(* CoDeSys 2.3.9.41 project: pns-dio.pro *)
(* Libraries: STANDARD.LIB 4.10.05 10:14:46, IECSFC.LIB 13.4.06 14:51:28, SYSLIBTIME.LIB 20.2.06 13:31:16, SYSTASKINFO.LIB 20.2.06 13:31:38, ANALYZATION.LIB 5.10.99 08:05:06, SYSLIBCALLBACK.LIB 20.2.06 13:31:08 *)

(* PLC configuration (modules and I/O channels)
AT %IB0.0 [ByteInput] 8 discrete inputs
DO0 AT %QX1.0 [BitOutput] relay
DO1 AT %QX2.0 [BitOutput] relay
DO2 AT %QX3.0 [BitOutput] relay
DO3 AT %QX4.0 [BitOutput] relay
DO4 AT %QX5.0 [BitOutput] relay
DO5 AT %QX6.0 [BitOutput] relay
AT %QX7.0 [BitOutput] Special output
RS-485-1 [COM1_USART] node 0, in %IB8.0.0 out %QB8.0.0 {CommunicationSpeed = 19200; Parity = NO PARITY CHECK; BitLength = 8 bits; StopLength = One stop bit; InterfaceType = RS485; FrameOriented = RTU; Timeout = 0; Visibility = No}
DIs AT %QW8.1.0 [WordOutput]
DOs AT %QW8.2.0 [WordOutput]
*)

(* POU PLC_PRG, ST *)
PROGRAM PLC_PRG
VAR
	NO_FIRST_PASS: BOOL := FALSE;
END_VAR
IF NO_FIRST_PASS = FALSE THEN
			DIs := 0;
			DOs := 0;
			DO0 := FALSE;
			DO1 := FALSE;
			DO2 := FALSE;
			DO3 := FALSE;
			DO4 := FALSE;
			DO5 := FALSE;
			NO_FIRST_PASS := TRUE;
END_IF;

DIs.0 := DI0;
DIs.1 := DI1;
DIs.2 := DI2;
DIs.3 := DI3;
DIs.4 := DI4;
DIs.5 := DI5;
DIs.6 := DI6;
DIs.7 := DI7;

DO0 := DOs.0;
DO1 := DOs.1;
DO2 := DOs.2;
DO3 := DOs.3;
DO4 := DOs.4;
DO5 := DOs.5;
END_PROGRAM
